INTERFACE I_Mc2Axis EXTENDS I_Component, I_AxisEnable, I_Mc2AxisRef, I_Resettable, I_Stoppable, I_AxisDynamics, I_AxisStatus, I_AxisJog, I_AxisHome, I_Mc2Settings

{attribute 'monitoring' := 'call'}
PROPERTY ErrorId : UDINT
GET
END_GET
END_PROPERTY

PROPERTY MotionTasks : I_MotionTaskCollection
GET
END_GET
END_PROPERTY

END_INTERFACE

(* stored: Version 1.1.0.1, ProductVersion 3.1.4026.20
   Itf I_Mc2Axis: Id {347e2aef-5611-452f-9ffc-b6ad926a510a}
   Property ErrorId: Id {d56d1c5d-53c1-4373-b824-480679d3561e}
   Get Get: Id {88d502ca-e062-4cb1-99bc-c31a0f99aa8c}
   Property MotionTasks: Id {6914240b-1882-4d81-a55f-46a091800bfd}
   Get Get: Id {526ff234-4916-45a3-8e29-4a9ed0e2f45f} *)
